{attribute 'pack_mode' := '8'} 
TYPE TableEntry :
STRUCT
    ID : LINT;
    JS : WSTRING(50);
    FTPBROWSE : BOOL;
    FTPDOWN : BOOL;
    DATAEXPORT : BOOL;
    DICTEDIT : BOOL;
    CREATETAB : BOOL;
END_STRUCT
END_TYPE;

(* stored: Version 1.1.0.1, ProductVersion 3.1.4024.16
   DUT TableEntry: Id {e0dd3824-7b69-4a86-81d3-7b5c20dc9f37} *)
